TYPE Y_YuklemeBaslatma :
STRUCT
END_STRUCT
END_TYPE

(* stored: Version 1.1.0.1, ProductVersion 3.1.4024.12
   DUT Y_YuklemeBaslatma: Id {ef40b6a0-fa93-4207-869d-7709ac902e93} *)
